PROGRAM P_Read_Research_Data
VAR


END_VAR

//***********************************************************************************
//
// ETH Zürich / Robotic Fabrication Lab
// HIB C 13 / Stefano-Franscini-Platz 1
// CH-8093 Zürich
// 
// ***********************************************************************************
// 
// PROJECT     :  A061 Inline Mixer
// 
// FUNCTION    :  Read all research data for the process
// 
// AUTHOR      :  Seyma Gürel / Philippe Fleischmann
// 
// EMAIL       :  scotto@arch.ethz.ch / fleischmann@arch.ehtz.ch
// 
// Copyright   :  ETH Zürich (CH) 2021
//
// ***********************************************************************************

// 
// Mode [] (0916 WT)
GVL_ResearchData.b_RED_Mode_Manual:= GVL_VAR.b_Mode_Manual;
GVL_ResearchData.b_RED_Mode_Laptop:= GVL_VAR.b_Mode_Laptop;

//
// Mixer run []
GVL_ResearchData.b_RED_Status_On:=GVL_VAR.b_MI1_Run;

//
// Mixer 1 speed override [%]
GVL_ResearchData.f_RED_Status_Speed_Overide:=GVL_VAR.f_MI1_Override;

//
// Mixer 1 current speed []
GVL_ResearchData.f_RED_Status_Speed_Motor_1:=GVL.Axis_Mixer1.NcToPlc.ActVelo;

//
// Mixer 1 current torque []
GVL_ResearchData.f_RED_Status_Torque_Motor_1:=GVL.f_MID1_ActTorque;

//
// Mixer 1 current motor temperature []
GVL_ResearchData.f_RED_Status_Temperature_Motor_1:=GVL.in_MID1_ActMotorTemperature *0.1; // weiting added 220817

//
// Mixer 2 current speed []
GVL_ResearchData.f_RED_Status_Speed_Motor_2:=GVL.Axis_Mixer1.NcToPlc.ActVelo;

//
// Mixer 2 current torque []
GVL_ResearchData.f_RED_Status_Torque_Motor_2:=GVL.f_MID2_ActTorque;

//
// Mixer 1 current motor temperature []
GVL_ResearchData.f_RED_Status_Temperature_Motor_2:=GVL.in_MID2_ActMotorTemperature *0.1; // weiting added 220817


// Superplasticizer maximum pump flowrate [ml/min]
GVL_ResearchData.f_RED_Status_Superplasticizer_Pump_Max_Flowrate_ml_per_min:=18.0;

//
// Accelration pump flowrate [ml/min]
GVL_ResearchData.f_RED_Status_Acceleration_Pump_Max_Flowrate_ml_per_min:=180.0;

END_PROGRAM

(* stored: Version 1.1.0.1, ProductVersion 3.1.4024.11
   POU P_Read_Research_Data: Id {affa89fd-b285-40f3-982b-c7fb6b079584}, SpecialFunc None *)
